# EPICS autosave request: softGlueApp/Db/ScalToStream8and16_settings.req
$(P)$(H)scalToStream-$(N)_desc
$(P)$(H)scalToStream-$(N)_CHADV_Signal
$(P)$(H)scalToStream-$(N)_ADVDONE_Signal
$(P)$(H)scalToStream-$(N)_FULL_Signal
$(P)$(H)scalToStream-$(N)_RESET_Signal
$(P)$(H)scalToStream-$(N)_DMAWORDS
$(P)$(H)scalToStream-$(N)_IMTRIG_Signal
$(P)$(H)scalToStream-$(N)_FLUSH_Signal
